FUNCTION_BLOCK AI_force
VAR_INPUT
	Raw_IO : INT;
END_VAR

VAR_OUTPUT
	Out : INT;
END_VAR

VAR
	ForceEnable : BOOL;
	ForceValue : INT;
END_VAR

IF NOT ForceEnable THEN
	OUT := Raw_IO;
ELSE
	OUT := ForceValue;
END_IF

END_FUNCTION_BLOCK

(* stored: Version 1.1.0.1, ProductVersion 3.1.4024.14
   POU AI_force: Id {e6fbe259-0513-417f-9edf-27f27c4a73bb}, SpecialFunc None *)
